FUNCTION Convert_UDINT_TO_BOOL : Hresult
VAR_INPUT
	in : UDINT;
	out : REFERENCE TO BOOL;
END_VAR
VAR
	converted : BOOL;
END_VAR
VAR CONSTANT
	INCOMPATIBLE : HRESULT := 16#9811070E;
END_VAR

converted := UDINT_TO_BOOL(in);

IF (BOOL_TO_UDINT(converted) <> in) THEN
	Convert_UDINT_TO_BOOL := INCOMPATIBLE;
	RETURN;
END_IF

out := converted;

END_FUNCTION

(* stored: Version 1.1.0.1, ProductVersion 3.1.4024.12
   POU Convert_UDINT_TO_BOOL: Id {6cc2dd0a-312e-42fd-90d2-65c72fb7a0fe}, SpecialFunc None *)
